LIN {X 0,Y 75.091,Z 921.072,A -85,B 0,C 180,E1 -30245.37,E2 -30245.37} C_VEL
LIN {X 0,Y 74.219,Z 922.443,A -85,B 0,C 180,E1 -30247.92,E2 -30247.92} C_VEL
LIN {X 0,Y 73.228,Z 923.726,A -85,B 0,C 180,E1 -30249.821,E2 -30249.821} C_VEL
LIN {X 0,Y 63.776,Z 931.104,A -85,B 0,C 180,E1 -30255.416,E2 -30255.416} C_VEL
LIN {X 0,Y 56.287,Z 936,A -85,B 0,C 180,E1 -30260.574,E2 -30260.574} C_VEL
LIN {X 0,Y 50.021,Z 939.546,A -85,B 0,C 180,E1 -30265.78,E2 -30265.78} C_VEL
LIN {X 0,Y 42.239,Z 943.122,A -85,B 0,C 180,E1 -30273.735,E2 -30273.735} C_VEL
LIN {X 0,Y 37.401,Z 945.144,A -85,B 0,C 180,E1 -30281.297,E2 -30281.297} C_VEL
LIN {X 0,Y 30.746,Z 947.896,A -85,B 0,C 180,E1 -30302.822,E2 -30302.822} C_VEL
LIN {X 0,Y 29.568,Z 948.694,A -85,B 0,C 180,E1 -30316.275,E2 -30316.275} C_VEL
LIN {X 0,Y 29.93,Z 949.075,A -85,B 0,C 180,E1 -30330.024,E2 -30330.024} C_VEL
LIN {X 0,Y 30.321,Z 948.275,A -85,B 0,C 180,E1 -30352.008,E2 -30352.008} C_VEL
LIN {X 0,Y 33.898,Z 946.74,A -85,B 0,C 180,E1 -30368.488,E2 -30368.488} C_VEL
LIN {X 0,Y 40.311,Z 944.222,A -85,B 0,C 180,E1 -30381.707,E2 -30381.707} C_VEL
LIN {X 0,Y 44.609,Z 942.438,A -85,B 0,C 180,E1 -30387.11,E2 -30387.11} C_VEL
LIN {X 0,Y 45.617,Z 941.525,A -85,B 0,C 180,E1 -30390.224,E2 -30390.224} C_VEL
LIN {X 0,Y 43.84,Z 935.865,A -85,B 0,C 180,E1 -30429.225,E2 -30429.225} C_VEL
LIN {X 0,Y 54.803,Z 931.288,A -85,B 0,C 180,E1 -30450.862,E2 -30450.862} C_VEL
LIN {X 0,Y 55.209,Z 931.302,A -85,B 0,C 180,E1 -30453.009,E2 -30453.009} C_VEL
LIN {X 0,Y 46.624,Z 935.076,A -85,B 0,C 180,E1 -30461.066,E2 -30461.066} C_VEL
LIN {X 0,Y 41.985,Z 936.862,A -85,B 0,C 180,E1 -30467.944,E2 -30467.944} C_VEL
LIN {X 0,Y 38,Z 938.201,A -85,B 0,C 180,E1 -30476.278,E2 -30476.278} C_VEL
LIN {X 0,Y 32.778,Z 939.753,A -85,B 0,C 180,E1 -30497.597,E2 -30497.597} C_VEL
LIN {X 0,Y 32.158,Z 939.959,A -85,B 0,C 180,E1 -30509.978,E2 -30509.978} C_VEL
LIN {X 0,Y 34.771,Z 939.213,A -85,B 0,C 180,E1 -30533.821,E2 -30533.821} C_VEL
LIN {X 0,Y 37.98,Z 938.263,A -85,B 0,C 180,E1 -30543.697,E2 -30543.697} C_VEL
LIN {X 0,Y 41.96,Z 936.951,A -85,B 0,C 180,E1 -30552.04,E2 -30552.04} C_VEL
LIN {X 0,Y 49.158,Z 934.159,A -85,B 0,C 180,E1 -30561.818,E2 -30561.818} C_VEL
LIN {X 0,Y 57.527,Z 930.302,A -85,B 0,C 180,E1 -30568.754,E2 -30568.754} C_VEL
LIN {X 0,Y 66.375,Z 925.363,A -85,B 0,C 180,E1 -30574.133,E2 -30574.133} C_VEL
LIN {X 0,Y 71.365,Z 922.101,A -85,B 0,C 180,E1 -30576.801,E2 -30576.801} C_VEL
LIN {X 0,Y 72.754,Z 920.79,A -85,B 0,C 180,E1 -30580.241,E2 -30580.241} C_VEL
LIN {X 0,Y 73.54,Z 919.994,A -85,B 0,C 180,E1 -30583.394,E2 -30583.394} C_VEL
LIN {X 0,Y 75.051,Z 918.737,A -85,B 0,C 180,E1 -30589.205,E2 -30589.205} C_VEL
LIN {X 0,Y 76.336,Z 918.05,A -85,B 0,C 180,E1 -30594.717,E2 -30594.717} C_VEL
LIN {X 0,Y 76.318,Z 918.456,A -85,B 0,C 180,E1 -30597.796,E2 -30597.796} C_VEL
LIN {X 0,Y 75.934,Z 919.076,A -85,B 0,C 180,E1 -30599.627,E2 -30599.627} C_VEL
LIN {X 0,Y 74.244,Z 920.834,A -85,B 0,C 180,E1 -30601.973,E2 -30601.973} C_VEL
LIN {X 0,Y 71.79,Z 922.968,A -85,B 0,C 180,E1 -30603.84,E2 -30603.84} C_VEL
LIN {X 0,Y 67.54,Z 926.26,A -85,B 0,C 180,E1 -30606.024,E2 -30606.024} C_VEL
LIN {X 0,Y 63.054,Z 929.402,A -85,B 0,C 180,E1 -30608.187,E2 -30608.187} C_VEL
LIN {X 0,Y 54.131,Z 934.914,A -85,B 0,C 180,E1 -30613.218,E2 -30613.218} C_VEL
LIN {X 0,Y 48.887,Z 937.696,A -85,B 0,C 180,E1 -30616.709,E2 -30616.709} C_VEL
LIN {X 0,Y 38.729,Z 942.074,A -85,B 0,C 180,E1 -30624.907,E2 -30624.907} C_VEL
LIN {X 0,Y 33.103,Z 944.09,A -85,B 0,C 180,E1 -30631.914,E2 -30631.914} C_VEL
LIN {X 0,Y 24.593,Z 946.845,A -85,B 0,C 180,E1 -30655.178,E2 -30655.178} C_VEL
LIN {X 0,Y 22.665,Z 947.641,A -85,B 0,C 180,E1 -30671.969,E2 -30671.969} C_VEL
LIN {X 0,Y 22.813,Z 948.03,A -85,B 0,C 180,E1 -30690.032,E2 -30690.032} C_VEL
LIN {X 0,Y 23.648,Z 947.299,A -85,B 0,C 180,E1 -30716.929,E2 -30716.929} C_VEL
LIN {X 0,Y 28.676,Z 945.696,A -85,B 0,C 180,E1 -30737.364,E2 -30737.364} C_VEL
LIN {X 0,Y 35.761,Z 943.374,A -85,B 0,C 180,E1 -30749.841,E2 -30749.841} C_VEL
LIN {X 0,Y 37.12,Z 942.426,A -85,B 0,C 180,E1 -30754.448,E2 -30754.448} C_VEL
LIN {X 0,Y 37.094,Z 938.16,A -85,B 0,C 180,E1 -30790.922,E2 -30790.922} C_VEL
LIN {X 0,Y 44.99,Z 935.1,A -85,B 0,C 180,E1 -30809.71,E2 -30809.71} C_VEL
LIN {X 0,Y 43.848,Z 935.559,A -85,B 0,C 180,E1 -30812.423,E2 -30812.423} C_VEL
LIN {X 0,Y 37.068,Z 937.894,A -85,B 0,C 180,E1 -30820.649,E2 -30820.649} C_VEL
LIN {X 0,Y 32.391,Z 939.233,A -85,B 0,C 180,E1 -30829.36,E2 -30829.36} C_VEL
LIN {X 0,Y 25.988,Z 940.781,A -85,B 0,C 180,E1 -30854.282,E2 -30854.282} C_VEL
LIN {X 0,Y 25.148,Z 940.989,A -85,B 0,C 180,E1 -30869.971,E2 -30869.971} C_VEL
LIN {X 0,Y 28.487,Z 940.244,A -85,B 0,C 180,E1 -30899.536,E2 -30899.536} C_VEL
LIN {X 0,Y 32.37,Z 939.294,A -85,B 0,C 180,E1 -30910.614,E2 -30910.614} C_VEL
LIN {X 0,Y 37.042,Z 937.981,A -85,B 0,C 180,E1 -30919.338,E2 -30919.338} C_VEL
LIN {X 0,Y 45.154,Z 935.189,A -85,B 0,C 180,E1 -30928.842,E2 -30928.842} C_VEL
LIN {X 0,Y 54.217,Z 931.332,A -85,B 0,C 180,E1 -30935.114,E2 -30935.114} C_VEL
LIN {X 0,Y 63.625,Z 926.392,A -85,B 0,C 180,E1 -30939.833,E2 -30939.833} C_VEL
LIN {X 0,Y 66.72,Z 924.485,A -85,B 0,C 180,E1 -30941.578,E2 -30941.578} C_VEL
LIN {X 0,Y 68.638,Z 923.152,A -85,B 0,C 180,E1 -30948.183,E2 -30948.183} C_VEL
LIN {X 0,Y 70.534,Z 922.319,A -85,B 0,C 180,E1 -30955.006,E2 -30955.006} C_VEL
LIN {X 0,Y 70.269,Z 923.308,A -85,B 0,C 180,E1 -30960.498,E2 -30960.498} C_VEL
LIN {X 0,Y 69.539,Z 924.285,A -85,B 0,C 180,E1 -30962.893,E2 -30962.893} C_VEL
LIN {X 0,Y 67.619,Z 926.197,A -85,B 0,C 180,E1 -30965.966,E2 -30965.966} C_VEL
LIN {X 0,Y 63.054,Z 929.402,A -85,B 0,C 180,E1 -30968.187,E2 -30968.187} C_VEL
LIN {X 0,Y 58.273,Z 932.316,A -85,B 0,C 180,E1 -30970.012,E2 -30970.012} C_VEL
LIN {X 0,Y 53.004,Z 934.913,A -85,B 0,C 180,E1 -30971.055,E2 -30971.055} C_VEL
LIN {X 0,Y 41.807,Z 939.222,A -85,B 0,C 180,E1 -30972.624,E2 -30972.624} C_VEL
LIN {X 0,Y 36.25,Z 941.055,A -85,B 0,C 180,E1 -30974.736,E2 -30974.736} C_VEL
LIN {X 0,Y 34.483,Z 941.611,A -85,B 0,C 180,E1 -30975.961,E2 -30975.961} C_VEL
LIN {X 0,Y 24.083,Z 944.611,A -85,B 0,C 180,E1 -30988.964,E2 -30988.964} C_VEL
LIN {X 0,Y 15.998,Z 946.588,A -85,B 0,C 180,E1 -31023.99,E2 -31023.99} C_VEL
LIN {X 0,Y 15.691,Z 946.984,A -85,B 0,C 180,E1 -31050.046,E2 -31050.046} C_VEL
LIN {X 0,Y 17.311,Z 946.308,A -85,B 0,C 180,E1 -31085.714,E2 -31085.714} C_VEL
LIN {X 0,Y 27.052,Z 943.968,A -85,B 0,C 180,E1 -31114.127,E2 -31114.127} C_VEL
LIN {X 0,Y 28.303,Z 943.63,A -85,B 0,C 180,E1 -31115.839,E2 -31115.839} C_VEL
LIN {X 0,Y 28.885,Z 943.005,A -85,B 0,C 180,E1 -31120.974,E2 -31120.974} C_VEL
LIN {X 0,Y 34.587,Z 938.456,A -85,B 0,C 180,E1 -31166.789,E2 -31166.789} C_VEL
LIN {X 0,Y 32.925,Z 938.926,A -85,B 0,C 180,E1 -31171.331,E2 -31171.331} C_VEL
LIN {X 0,Y 27.443,Z 940.265,A -85,B 0,C 180,E1 -31179.76,E2 -31179.76} C_VEL
LIN {X 0,Y 19.342,Z 941.809,A -85,B 0,C 180,E1 -31208.655,E2 -31208.655} C_VEL
LIN {X 0,Y 18.137,Z 942.018,A -85,B 0,C 180,E1 -31229.96,E2 -31229.96} C_VEL
LIN {X 0,Y 22.642,Z 941.275,A -85,B 0,C 180,E1 -31268.333,E2 -31268.333} C_VEL
LIN {X 0,Y 27.42,Z 940.325,A -85,B 0,C 180,E1 -31280.216,E2 -31280.216} C_VEL
LIN {X 0,Y 32.899,Z 939.012,A -85,B 0,C 180,E1 -31288.661,E2 -31288.661} C_VEL
LIN {X 0,Y 41.953,Z 936.22,A -85,B 0,C 180,E1 -31297.081,E2 -31297.081} C_VEL
LIN {X 0,Y 51.656,Z 932.362,A -85,B 0,C 180,E1 -31302.199,E2 -31302.199} C_VEL
LIN {X 0,Y 58.254,Z 929.175,A -85,B 0,C 180,E1 -31304.778,E2 -31304.778} C_VEL
LIN {X 0,Y 61.789,Z 927.307,A -85,B 0,C 180,E1 -31306.851,E2 -31306.851} C_VEL
LIN {X 0,Y 63.9,Z 926.425,A -85,B 0,C 180,E1 -31313.685,E2 -31313.685} C_VEL
LIN {X 0,Y 63.916,Z 927.224,A -85,B 0,C 180,E1 -31320,E2 -31320} C_VEL
LIN {X 0,Y 63.247,Z 927.762,A -85,B 0,C 180,E1 -31320.929,E2 -31320.929} C_VEL
LIN {X 0,Y 52.929,Z 933.826,A -85,B 0,C 180,E1 -31325.373,E2 -31325.373} C_VEL
LIN {X 0,Y 42.878,Z 938.552,A -85,B 0,C 180,E1 -31330.538,E2 -31330.538} C_VEL
LIN {X 0,Y 34.483,Z 941.611,A -85,B 0,C 180,E1 -31335.961,E2 -31335.961} C_VEL
LIN {X 0,Y 29.148,Z 943.106,A -85,B 0,C 180,E1 -31339.728,E2 -31339.728} C_VEL
LIN {X 0,Y 19.751,Z 944.721,A -85,B 0,C 180,E1 -31346.287,E2 -31346.287} C_VEL
LIN {X 0,Y 12.558,Z 945.43,A -85,B 0,C 180,E1 -31358.405,E2 -31358.405} C_VEL
LIN {X 0,Y 8.814,Z 945.76,A -85,B 0,C 180,E1 -31383.522,E2 -31383.522} C_VEL
LIN {X 0,Y 8.418,Z 945.824,A -85,B 0,C 180,E1 -31396.386,E2 -31396.386} C_VEL
LIN {X 0,Y 8.565,Z 945.938,A -85,B 0,C 180,E1 -31410.084,E2 -31410.084} C_VEL
LIN {X 0,Y 15.406,Z 944.764,A -85,B 0,C 180,E1 -31475.947,E2 -31475.947} C_VEL
LIN {X 0,Y 20.091,Z 943.924,A -85,B 0,C 180,E1 -31484.279,E2 -31484.279} C_VEL
LIN {X 0,Y 21.253,Z 943.222,A -85,B 0,C 180,E1 -31493.032,E2 -31493.032} C_VEL
LIN {X 0,Y 24.343,Z 941.281,A -85,B 0,C 180,E1 -31521.133,E2 -31521.133} C_VEL
LIN {X 0,Y 23.576,Z 941.297,A -85,B 0,C 180,E1 -31526.515,E2 -31526.515} C_VEL
LIN {X 0,Y 13.071,Z 942.837,A -85,B 0,C 180,E1 -31557.408,E2 -31557.408} C_VEL
LIN {X 0,Y 11.124,Z 943.047,A -85,B 0,C 180,E1 -31589.935,E2 -31589.935} C_VEL
LIN {X 0,Y 13.054,Z 942.862,A -85,B 0,C 180,E1 -31622.507,E2 -31622.507} C_VEL
LIN {X 0,Y 23.551,Z 941.356,A -85,B 0,C 180,E1 -31653.471,E2 -31653.471} C_VEL
LIN {X 0,Y 29.854,Z 940.043,A -85,B 0,C 180,E1 -31660.258,E2 -31660.258} C_VEL
LIN {X 0,Y 39.747,Z 937.25,A -85,B 0,C 180,E1 -31666.45,E2 -31666.45} C_VEL
LIN {X 0,Y 49.958,Z 933.392,A -85,B 0,C 180,E1 -31669.892,E2 -31669.892} C_VEL
LIN {X 0,Y 56.763,Z 930.259,A -85,B 0,C 180,E1 -31671.997,E2 -31671.997} C_VEL
LIN {X 0,Y 57.635,Z 930.021,A -85,B 0,C 180,E1 -31674.598,E2 -31674.598} C_VEL
LIN {X 0,Y 56.339,Z 930.859,A -85,B 0,C 180,E1 -31676.126,E2 -31676.126} C_VEL
LIN {X 0,Y 46.374,Z 935.737,A -85,B 0,C 180,E1 -31679.319,E2 -31679.319} C_VEL
LIN {X 0,Y 38.663,Z 938.81,A -85,B 0,C 180,E1 -31681.957,E2 -31681.957} C_VEL
LIN {X 0,Y 28.278,Z 941.988,A -85,B 0,C 180,E1 -31686.442,E2 -31686.442} C_VEL
LIN {X 0,Y 15.209,Z 944.738,A -85,B 0,C 180,E1 -31702.576,E2 -31702.576} C_VEL
LIN {X 0,Y 8.418,Z 945.824,A -85,B 0,C 180,E1 -31756.386,E2 -31756.386} C_VEL
LIN {X 0,Y 7.431,Z 945.715,A -85,B 0,C 180,E1 -31756.402,E2 -31756.402} C_VEL
LIN {X 0,Y 5.953,Z 945.41,A -85,B 0,C 180,E1 -31740.093,E2 -31740.093} C_VEL
LIN {X 0,Y 6.096,Z 944.968,A -85,B 0,C 180,E1 -31706.671,E2 -31706.671} C_VEL
LIN {X 0,Y 13.062,Z 943.726,A -85,B 0,C 180,E1 -31671.145,E2 -31671.145} C_VEL
LIN {X 0,Y 17.795,Z 942.972,A -85,B 0,C 180,E1 -31668.868,E2 -31668.868} C_VEL
LIN {X 0,Y 19.688,Z 942.618,A -85,B 0,C 180,E1 -31669.626,E2 -31669.626} C_VEL
LIN {X 0,Y 21.359,Z 942.388,A -85,B 0,C 180,E1 -31670.59,E2 -31670.59} C_VEL
LIN {X 0,Y 21.241,Z 942.506,A -85,B 0,C 180,E1 -31672.74,E2 -31672.74} C_VEL
LIN {X 0,Y 7.016,Z 944.488,A -85,B 0,C 180,E1 -31680.558,E2 -31680.558} C_VEL
LIN {X 0,Y 1.418,Z 944.889,A -85,B 0,C 180,E1 -31770.508,E2 -31770.508} C_VEL
LIN {X 0,Y 14.094,Z 943.717,A -85,B 0,C 180,E1 -31863.459,E2 -31863.459} C_VEL
LIN {X 0,Y 14.568,Z 943.286,A -85,B 0,C 180,E1 -31875.044,E2 -31875.044} C_VEL
LIN {X 0,Y 4.11,Z 944.077,A -85,B 0,C 180,E1 -31949.825,E2 -31949.825} C_VEL
LIN {X 0,Y 8.076,Z 943.89,A -85,B 0,C 180,E1 -32010.298,E2 -32010.298} C_VEL
LIN {X 0,Y 19.688,Z 942.618,A -85,B 0,C 180,E1 -32029.626,E2 -32029.626} C_VEL
LIN {X 0,Y 19.688,Z 942.618,A -85,B 0,C 180,E1 -32029.626,E2 -32029.626}

QRS_NEXT_CUT()

QRS_NEXT()
QRS_HOME()

END
